// TIA Portal V17 export
// export: Created 2022-07-20T07:01:31.5853056Z, ExportSetting WithDefaults, DisplayName Totally Integrated Automation Portal, DisplayVersion V17, DisplayName TIA Portal Openness, DisplayVersion V17, DisplayName TIA Portal Version Control Interface, DisplayVersion V17, DisplayName SINAMICS Startdrive Advanced, DisplayVersion V17, DisplayName SINAMICS Startdrive G130, G150, S120, S150, SINAMICS MV, S210, DisplayVersion V17, DisplayName SINAMICS Startdrive G110M, G120, G120C, G120D, G120P, G115D, DisplayVersion V17, DisplayName STEP 7 Professional, DisplayVersion V17, DisplayName STEP 7 Safety, DisplayVersion V17, DisplayName WinCC Advanced, DisplayVersion V17
FUNCTION "FC10331_UDintTo4Bytes" : Void   // FC10331, LAD
{ S7_Optimized_Access := 'TRUE' }
VERSION : 0.1
// stored: AutoNumber false, IsIECCheckEnabled false, SetENOAutomatically false, UDAEnableTagReadback false
   VAR_INPUT
      UDint : UDInt;
   END_VAR
   VAR_OUTPUT
      Byte_0 : Byte;
      Byte_1 : Byte;
      Byte_2 : Byte;
      Byte_3 : Byte;
   END_VAR
BEGIN

REGION Network 1 (SCL)
   #Byte_0.%X0 := #UDint.%X0;
   #Byte_0.%X1 := #UDint.%X1;
   #Byte_0.%X2 := #UDint.%X2;
   #Byte_0.%X3 := #UDint.%X3;
   #Byte_0.%X4 := #UDint.%X4;
   #Byte_0.%X5 := #UDint.%X5;
   #Byte_0.%X6 := #UDint.%X6;
   #Byte_0.%X7 := #UDint.%X7;

   #Byte_1.%X0 := #UDint.%X8;
   #Byte_1.%X1 := #UDint.%X9;
   #Byte_1.%X2 := #UDint.%X10;
   #Byte_1.%X3 := #UDint.%X11;
   #Byte_1.%X4 := #UDint.%X12;
   #Byte_1.%X5 := #UDint.%X13;
   #Byte_1.%X6 := #UDint.%X14;
   #Byte_1.%X7 := #UDint.%X15;

   #Byte_2.%X0 := #UDint.%X16;
   #Byte_2.%X1 := #UDint.%X17;
   #Byte_2.%X2 := #UDint.%X18;
   #Byte_2.%X3 := #UDint.%X19;
   #Byte_2.%X4 := #UDint.%X20;
   #Byte_2.%X5 := #UDint.%X21;
   #Byte_2.%X6 := #UDint.%X22;
   #Byte_2.%X7 := #UDint.%X23;

   #Byte_3.%X0 := #UDint.%X24;
   #Byte_3.%X1 := #UDint.%X25;
   #Byte_3.%X2 := #UDint.%X26;
   #Byte_3.%X3 := #UDint.%X27;
   #Byte_3.%X4 := #UDint.%X28;
   #Byte_3.%X5 := #UDint.%X29;
   #Byte_3.%X6 := #UDint.%X30;
   #Byte_3.%X7 := #UDint.%X31;
END_REGION
END_FUNCTION
